// TIA Portal V20 export
TYPE "UDT_Service_StepOrder"
   STRUCT
      stepNumber : Int := -1;   // actual number of step
      stepMonitoringTime : UDInt := 1000;   // step monitoring time
      parameter : "UDT_Service_IndexElement";   // start index of used parameters in parameter Array
   END_STRUCT;
END_TYPE
